(* CODESYS project IO_Management.export

Project tree, tasks and I/O mapping:
  IO_Management/
    function block Digital_Input [ST]
    function block Digital_Input_Analog [ST]
    function block Digital_Output [ST]
*)

// IO_Management/Digital_Input
FUNCTION_BLOCK Digital_Input
VAR_INPUT
	enable : BOOL;
END_VAR
VAR_OUTPUT
	DI_Array : ARRAY [1..12] OF BOOL;
	DI_01 : BOOL;
	DI_02 : BOOL;
	DI_03 : BOOL;
	DI_04 : BOOL;
	DI_05 : BOOL;
	DI_06 : BOOL;
	DI_07 : BOOL;
	DI_08 : BOOL;
	DI_09 : BOOL;
	DI_10 : BOOL;
	DI_11 : BOOL;
	DI_12 : BOOL;
	DI_13 : BOOL;
	DI_14 : BOOL;
	DI_15 : BOOL;
	DI_16 : BOOL;
	DI_17 : BOOL;
	DI_18 : BOOL;
	DI_19 : BOOL;
	DI_20 : BOOL;
	DI_21 : BOOL;
	DI_22 : BOOL;
	DI_23 : BOOL;
	DI_24 : BOOL;
END_VAR
VAR
	forCounter: INT;
	
	Read_6Ax_DI: Arcalibrary.ECAT_GetPdi_U32;
	DI_Raw : UDINT;
END_VAR

// read di
Read_6Ax_DI(Enable:= enable, Offset:=143, Value=>DI_Raw);

// judge which bit is true
FOR forCounter := 1 TO UINT_TO_INT(SIZEOF(DI_Array)) DO // loop all bool value
	DI_Array[forCounter] := UDINT_TO_BOOL(DI_Raw AND SHL(1, forCounter - 1));
END_FOR

DI_01 := DI_Array[01];
DI_02 := DI_Array[02];
DI_03 := DI_Array[03];
DI_04 := DI_Array[04];
DI_05 := DI_Array[05];
DI_06 := DI_Array[06];
DI_07 := DI_Array[07];
DI_08 := DI_Array[08];
DI_09 := DI_Array[09];
DI_10 := DI_Array[10];
DI_11 := DI_Array[11];
DI_12 := DI_Array[12];
(*	// not yet ready, need add more code for second driver for more input
DI_13 := DI_Array[13];
DI_14 := DI_Array[14];
DI_15 := DI_Array[15];
DI_16 := DI_Array[16];
DI_17 := DI_Array[17];
DI_18 := DI_Array[18];
DI_19 := DI_Array[19];
DI_20 := DI_Array[20];
DI_21 := DI_Array[21];
DI_22 := DI_Array[22];
DI_23 := DI_Array[23];
DI_24 := DI_Array[24];
*)

END_FUNCTION_BLOCK

// IO_Management/Digital_Input_Analog
FUNCTION_BLOCK Digital_Input_Analog
VAR_INPUT
	enable : BOOL;
	MaxRawInputValue : ARRAY[0..7] OF UINT;
	MinRawInputValue :  ARRAY[0..7] OF UINT;
	MaxmentOffset : UINT := 50;
	SmoothTIme : TIME := T#200MS;
END_VAR
VAR_OUTPUT
	DIA_raw: ARRAY[0..7] OF UINT;
	DIA_Process : ARRAY[0..7] OF REAL;
END_VAR
VAR
	_Timer : ton;
	_sample_times : UINT;
	
	_DA: Arcalibrary.ECAT_GetPdi_U16;
	_offset : ARRAY[0..7] OF WORD;
	_raw_value : ARRAY[0..7] OF UDINT;
END_VAR

_offset[0]:=147;
_DA(enable:= enable, offset := _offset[0]);

_Timer(in:= TRUE, pt := SmoothTime);
_raw_value[0] := _raw_value[0] + _DA.Value;
_sample_times := _sample_times + 1;
IF _Timer.Q THEN
	DIA_raw[0] := UDINT_TO_UINT(_raw_value[0] / UINT_TO_UDINT(_sample_times));
	_raw_value[0] := 0;
	_sample_times := 0;
	_Timer (in := FALSE);
END_IF

DIA_Process[0] := (UINT_TO_REAL(DIA_raw[0])/UINT_TO_REAL((MaxRawInputValue[0] - MinRawInputValue[0]) - MaxmentOffset))*100;

IF DIA_Process[0] > 100 THEN
	DIA_Process[0] := 100;
END_IF

IF DIA_Process[0] < 0 THEN
	DIA_Process[0] := 0;
END_IF

END_FUNCTION_BLOCK

// IO_Management/Digital_Output
FUNCTION_BLOCK Digital_Output
VAR_INPUT
	enable : BOOL;
	DO_Array: ARRAY [1..8] OF BOOL;
	DO_01 : BOOL;
	DO_02 : BOOL;
	DO_03 : BOOL;
	DO_04 : BOOL;
	DO_05 : BOOL;
	DO_06 : BOOL;
	DO_07 : BOOL;
	DO_08 : BOOL;
END_VAR
VAR_OUTPUT
END_VAR
VAR
	forCounter: INT;
	
	Set_Do: ARRAY [1..8] OF BOOL;
	new_Do_Value, old_Do_Value : UINT;
	Write_6Ax_Do: Arcalibrary.ECAT_SetPdo_U32;
END_VAR

// write do
new_Do_Value:= 0;	// initialize 
Set_Do[01] := DO_Array[01] OR do_01;
Set_Do[02] := DO_Array[02] OR do_02;
Set_Do[03] := DO_Array[03] OR do_03;
Set_Do[04] := DO_Array[04] OR do_04;
Set_Do[05] := DO_Array[05] OR do_05;
Set_Do[06] := DO_Array[06] OR do_06;
Set_Do[07] := DO_Array[07] OR do_07;
Set_Do[08] := DO_Array[08] OR do_08;

// shift mamary according to bool
FOR forCounter := 1 TO UINT_TO_INT(SIZEOF(Set_Do)) DO // loop all bool value
	IF DO_Array[forCounter] THEN	// if out put is true
		new_Do_Value := new_Do_Value + SHL(1, forCounter - 1);
	END_IF
END_FOR

IF new_Do_Value <> old_Do_Value THEN
	old_Do_Value := new_Do_Value;
END_IF
Write_6Ax_Do(Enable:= enable, Offset:=143, Value:=old_Do_Value);	// write DO

END_FUNCTION_BLOCK
